FUNCTION_BLOCK MachineModes
VAR
	
	m_ptrServices: POINTER TO ServiceContainer;
	m_ptrPanelMgr: POINTER TO PanelManager;	
	m_path_File:STRING;
	m_stratState: EOperationResult;
	m_allFinished: BOOL;
	m_ton: TON;
	
	//testLog: FB_TimeLog;
	i: ULINT;
END_VAR

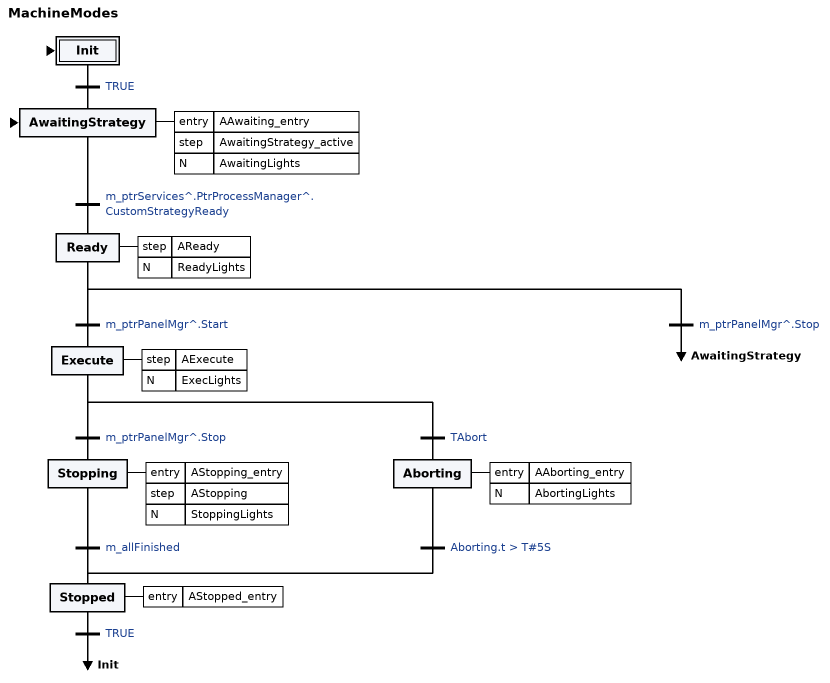
INITIAL_STEP Init:
END_STEP
TRANSITION FROM Init TO AwaitingStrategy
    := TRUE;
END_TRANSITION
STEP AwaitingStrategy:
    AAwaiting_entry(P1);  // entry action
    AwaitingStrategy_active(N);  // step action
    AwaitingLights(N);
END_STEP
TRANSITION FROM AwaitingStrategy TO Ready
    := m_ptrServices^.PtrProcessManager^.CustomStrategyReady;
END_TRANSITION
STEP Ready:
    AReady(N);  // step action
    ReadyLights(N);
END_STEP
TRANSITION FROM Ready TO Execute
    := m_ptrPanelMgr^.Start;
END_TRANSITION
TRANSITION FROM Ready TO AwaitingStrategy
    := m_ptrPanelMgr^.Stop;
END_TRANSITION
STEP Execute:
    AExecute(N);  // step action
    ExecLights(N);
END_STEP
TRANSITION FROM Execute TO Stopping
    := m_ptrPanelMgr^.Stop;
END_TRANSITION
STEP Stopping:
    AStopping_entry(P1);  // entry action
    AStopping(N);  // step action
    StoppingLights(N);
END_STEP
TRANSITION FROM Stopping TO Stopped
    := m_allFinished;
END_TRANSITION
TRANSITION FROM Execute TO Aborting
    := TAbort;
END_TRANSITION
STEP Aborting:
    AAborting_entry(P1);  // entry action
    AbortingLights(N);
END_STEP
TRANSITION FROM Aborting TO Stopped
    := Aborting.t > T#5S;
END_TRANSITION
STEP Stopped:
    AStopped_entry(P1);  // entry action
END_STEP
TRANSITION FROM Stopped TO Init
    := TRUE;
END_TRANSITION

ACTION AAborting_entry:
m_ptrServices^.PtrProcessManager^.RequestAbort();
m_ptrServices^.PtrErrorManager^.AddMessage(EAlarms.aborting, TRUE, ESeverity.info, 'Main');
END_ACTION

ACTION AAwaiting_entry:
m_ptrServices^.PtrErrorManager^.AddMessage(EAlarms.initialized, TRUE, ESeverity.info, 'Main');
END_ACTION

ACTION AbortingLights:
m_ptrPanelMgr^.SetGreen(FALSE);
m_ptrPanelMgr^.SetRed(TRUE, T#200MS);
m_ptrPanelMgr^.SetWhite(FALSE);
END_ACTION

ACTION AExecute:
//START_MESSUNG1
//testLog(bEnable := TRUE,bMeasureCode := TRUE, sFileName := m_path_File,);
m_stratState := m_ptrServices^.PtrProcessManager^.ExecuteCustomStrategy();
//ENDE_MESSUNG1
//testLog(bEnable := TRUE,bMeasureCode := FALSE, sFileName := m_path_File,);
END_ACTION

ACTION AReady:
// TODO - blink light or something...
END_ACTION

ACTION AStopped_entry:
m_ptrServices^.PtrProcessManager^.ResetConfiguration();
m_ptrServices^.PtrStateTracker^.ResetConfiguration();
m_ptrServices^.PtrErrorManager^.AddMessage(EAlarms.stopped, TRUE, ESeverity.info, 'Main');
END_ACTION

ACTION AStopping:
m_allFinished := m_ptrServices^.PtrProcessManager^.FinishPrimitives(TRUE);
END_ACTION

ACTION AStopping_entry:
m_ptrServices^.PtrErrorManager^.AddMessage(EAlarms.stopping, TRUE, ESeverity.info, 'Main');
END_ACTION

ACTION AwaitingLights:
m_ptrPanelMgr^.SetGreen(FALSE);
m_ptrPanelMgr^.SetRed(FALSE);
m_ptrPanelMgr^.SetWhite(TRUE, T#500MS);
END_ACTION

ACTION AwaitingStrategy_active:

END_ACTION

ACTION ExecLights:
m_ptrPanelMgr^.SetGreen(TRUE);
m_ptrPanelMgr^.SetRed(FALSE);
m_ptrPanelMgr^.SetWhite(FALSE);
END_ACTION

//FB_Init is always available implicitly and it is used primarily for initialization.
//The return value is not evaluated. For a specific influence, you can also declare the
//methods explicitly and provide additional code there with the standard initialization
//code. You can evaluate the return value.
METHOD FB_Init: BOOL
VAR_INPUT
    bInitRetains: BOOL; // TRUE: the retain variables are initialized (reset warm / reset cold)
    bInCopyCode: BOOL;  // TRUE: the instance will be copied to the copy code afterward (online change)
	
	i_ptrServices: POINTER TO ServiceContainer;
	i_ptrPanelMgr: POINTER TO PanelManager;	
	i_path_File:String;
END_VAR
VAR
	i: UINT;
	m_statesEnum: EProcessVariables;
END_VAR
m_ptrServices := i_ptrServices;
m_ptrPanelMgr := i_ptrPanelMgr;

// the panel manager serves as an observation of the buttons
m_ptrServices^.PtrStateTracker^.AddObservation(m_ptrPanelMgr);

// optionally, disable pre-/ postconditions
// m_ptrServices^.PtrProcessManager^.SetAllConditionsTrue();

// init process variable names
FOR i := ResiConst.ARR_MIN TO ResiConst.STATE_ARR_MAX DO
	m_statesEnum := i;
	i_ptrServices^.PtrStateTracker^.SetProcessVariableName(i, TO_STRING(m_statesEnum));
END_FOR

m_path_File:=i_path_File;
FC_InitAlarmTexts();
END_METHOD

ACTION ReadyLights:
m_ptrPanelMgr^.SetGreen(TRUE, T#500MS);
m_ptrPanelMgr^.SetRed(FALSE);
m_ptrPanelMgr^.SetWhite(FALSE);
END_ACTION

ACTION StoppingLights:
m_ptrPanelMgr^.SetGreen(FALSE);
m_ptrPanelMgr^.SetRed(TRUE, T#500MS);
m_ptrPanelMgr^.SetWhite(FALSE);
END_ACTION

TRANSITION TAbort:
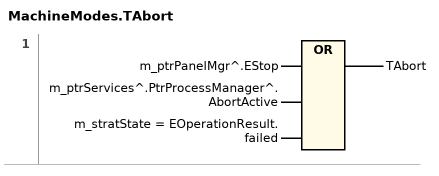
// NETWORK 1
TAbort := m_ptrPanelMgr^.EStop OR m_ptrServices^.PtrProcessManager^.AbortActive OR (m_stratState = EOperationResult.failed);
END_TRANSITION

END_FUNCTION_BLOCK

(* stored: Version 1.1.0.1
   POU MachineModes: Id {699dc84f-9b7c-4a66-84a1-3d4ea0291fad}, SpecialFunc None
   Folder PanelLights: Id {2794be32-3d1b-40b6-9715-d947a2db78cc}
   Action AAborting_entry: Id {aabbe950-c299-4669-9f98-abbb3c074288}
   Action AAwaiting_entry: Id {04c9d2f9-024a-4f35-b8cd-d84e65c58826}
   Action AbortingLights: Id {40bca023-17c1-4e53-a14a-1a033135acdd}
   Action AExecute: Id {21ef47d2-ac09-4936-91f0-e5b8a59695b2}
   Action AReady: Id {438ee1e7-7c7d-4cde-bbd5-8778170b23ae}
   Action AStopped_entry: Id {371d6257-40b5-4ccf-a20a-89f933968770}
   Action AStopping: Id {c2757091-41eb-49b3-90a6-52a4f9934378}
   Action AStopping_entry: Id {f1458812-e379-4750-b1af-3294fe7a82ec}
   Action AwaitingLights: Id {3cad2775-bea7-4c4b-852f-c1de3010631f}
   Action AwaitingStrategy_active: Id {84e601d7-b828-421d-8a57-28876b3f8872}
   Action ExecLights: Id {aa49f023-0d6b-4ff3-92cf-44df32f2f5a5}
   Method FB_init: Id {fbe1f0ff-3696-4599-9412-c7729cbd3ba8}
   Action ReadyLights: Id {b27533b3-9c17-4db6-bbe2-c44e67a39489}
   Action StoppingLights: Id {fdad32f2-2f4c-4b81-9c64-e0ced315c8fa}
   Transition TAbort: Id {bf8c27ad-c080-488f-b58a-9e4facb0e592} *)
